FUNCTION_BLOCK EnhancedAdapterWith2 (* FB for testing an adapter WITH connection *)
  (* Standard: 61499-2; Description: Copyright (c) 2023 Johannes Kepler University Linz This program and the accompanying materials are made available under the terms of the Eclipse Public License 2.0 which is available at https://www.eclipse.org/legal/epl-2.0/ SPDX-License-Identifier: EPL-2.0 *)
  (* Version 1.0, 2023-03-07, Bianca Wiesmayr, Johannes Kepler University Linz, initial API and implementation and/or initial documentation *)
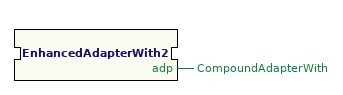
  PLUGS
    adp : CompoundAdapterWith;
  END_PLUGS
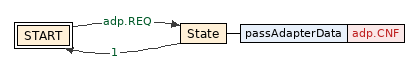
  EC_STATES
    START; (* Initial State *)
    State : passAdapterData -> adp.CNF;
  END_STATES
  EC_TRANSITIONS
    START TO State := adp.REQ;
    State TO START := 1;
  END_TRANSITIONS
  ALGORITHM passAdapterData IN ST:
	adp.DO1 := adp.DI1;
	adp.DO2 := adp.DI2;
  END_ALGORITHM
END_FUNCTION_BLOCK
